Fanuc KAREL source: kt00415.KL

-- PROVISIONAL review KL for V1013-1; original PC SHA256 3af2d0927ad053bec6fdc9e0a51509e6ed0569c76a0e1be99ad58a338d71608c
-- Incomplete behavior may be omitted. Consult companion uncertainty JSON. Do not deploy.
PROGRAM KT00415
%NOLOCKGROUP
VAR
  I2 : INTEGER
  OUT : BOOLEAN
-- UNRESOLVED_DECL H1 type=002017
BEGIN
  -- UNRESOLVED_PC offsets 5-19; opcodes 2E,22,9D,33,B4
  -- UNRESOLVED_PC offsets 24-35; opcodes 2E,23
  -- UNRESOLVED_PC offsets 40-62; opcodes 22,9D,33,B3,21,5B,23
  -- UNRESOLVED_PC offsets 67-71; opcodes 7F
END KT00415
